FUNCTION_BLOCK FB_System_DLK_951
VAR_INPUT
	Freigabe_auto				: BOOL;
	Freigabe_Deakt_auto			: BOOL;
	Betrieb_Anford_auto			: BOOL;
END_VAR
VAR_OUTPUT
	{attribute 'OPC.UA.DA' := '1'}Steuerung				: ST_System_DLK_Steuerung;		
	{attribute 'OPC.UA.DA' := '1'}Stellwert				: ST_System_DLK_Stellwert;		
	{attribute 'OPC.UA.DA' := '1'}Zustand					: ST_System_DLK_Zustand;	
	{attribute 'OPC.UA.DA' := '1'}Parameter				: ST_System_DLK_Parameter;		
END_VAR
VAR
	Pumpe_251				: FB_PU;
	Stellventil_251			: FB_SVs;
	Regelventil_251			: FB_RV;	(* 14.07.2020*)
	Druckluftkompressor_951	: FB_DLK;

	Zustandscheck			: FB_System_DLK_Zustandscheck;
	Logik					: FB_System_DLK_Logik;
	Ablaufsteuerung			: FB_System_DLK_Ablaufsteuerung;
	Stellwertscheck			: FB_System_DLK_Stellwertscheck;

END_VAR
VAR // added by the converter: edge detectors and wires of the graphical bodies
    _w1 : ANY;
END_VAR

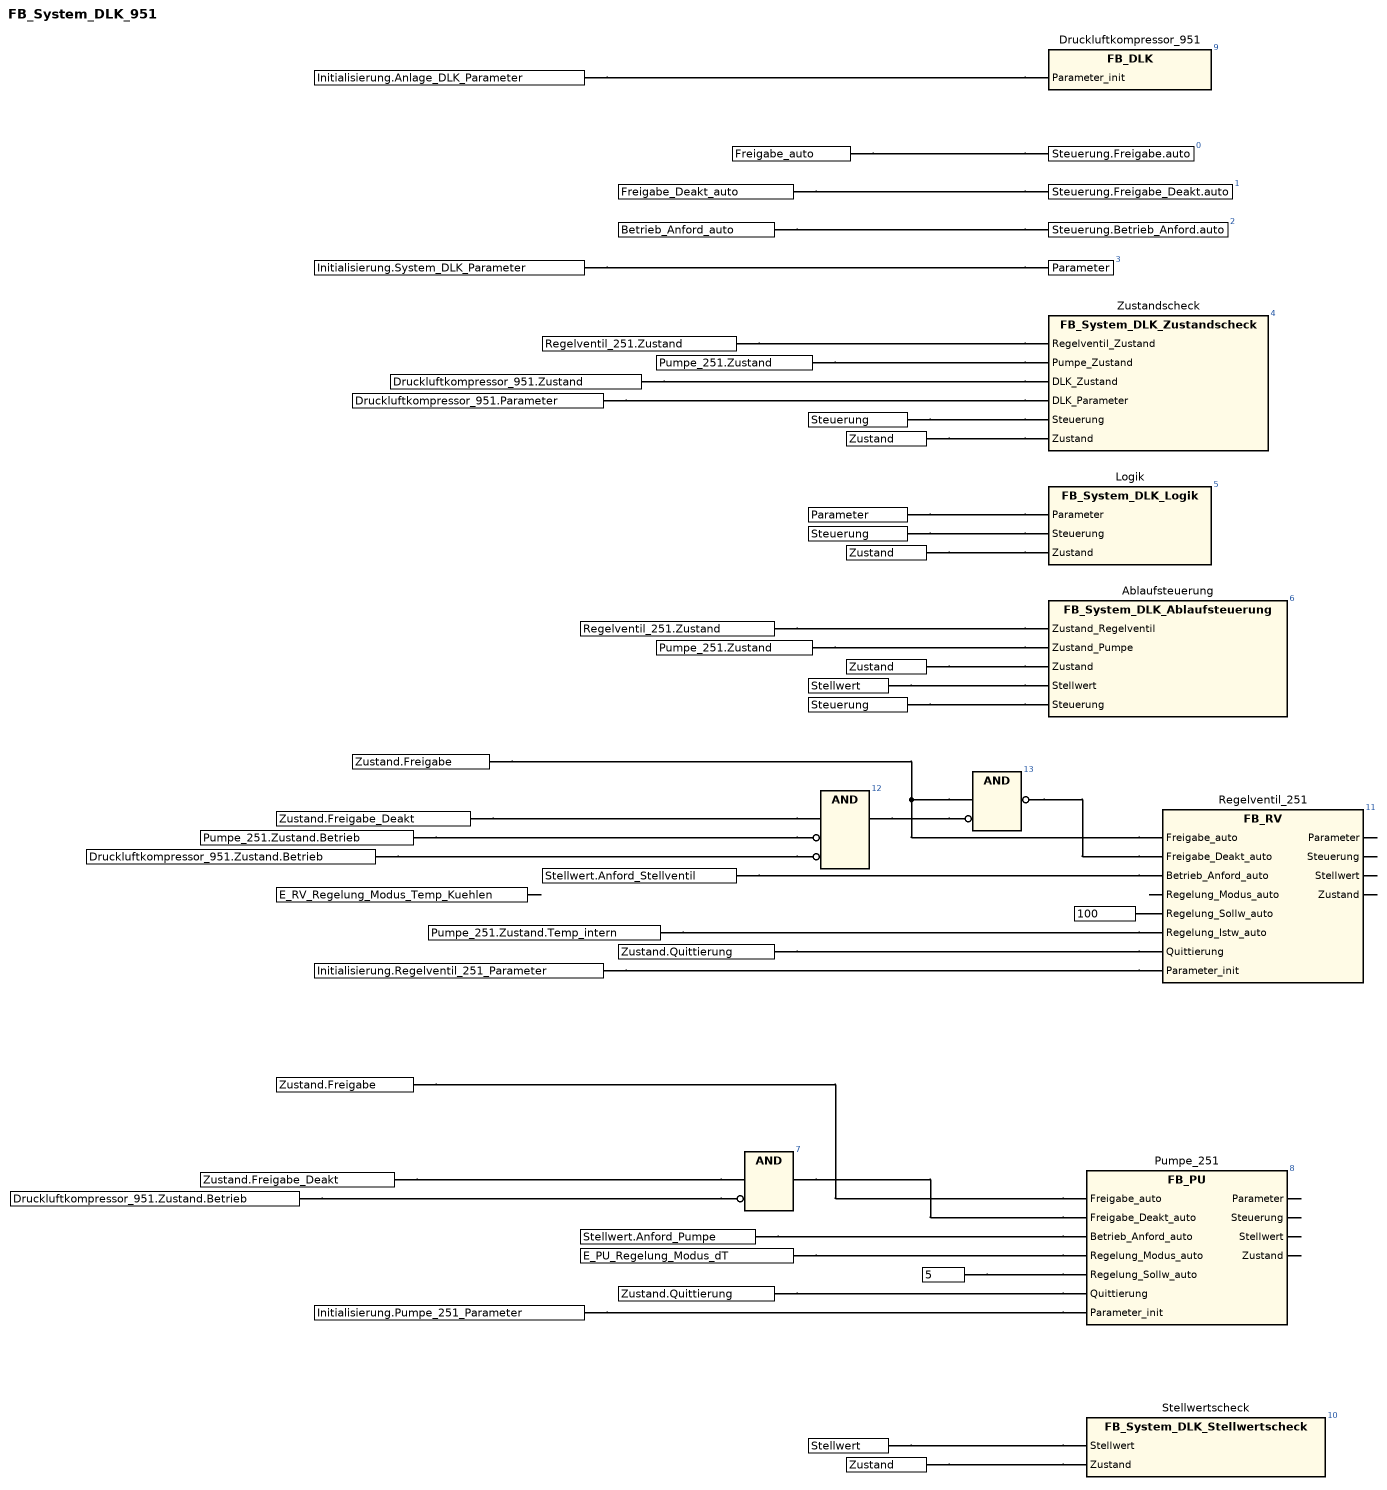
Steuerung.Freigabe.auto := Freigabe_auto;
Steuerung.Freigabe_Deakt.auto := Freigabe_Deakt_auto;
Steuerung.Betrieb_Anford.auto := Betrieb_Anford_auto;
Parameter := Initialisierung.System_DLK_Parameter;
Zustandscheck(
    Regelventil_Zustand := Regelventil_251.Zustand,
    Pumpe_Zustand := Pumpe_251.Zustand,
    DLK_Zustand := Druckluftkompressor_951.Zustand,
    DLK_Parameter := Druckluftkompressor_951.Parameter,
    Steuerung := Steuerung,
    Zustand := Zustand); // FB_System_DLK_Zustandscheck
Logik(Parameter := Parameter, Steuerung := Steuerung, Zustand := Zustand); // FB_System_DLK_Logik
Ablaufsteuerung(
    Zustand_Regelventil := Regelventil_251.Zustand,
    Zustand_Pumpe := Pumpe_251.Zustand,
    Zustand := Zustand,
    Stellwert := Stellwert,
    Steuerung := Steuerung); // FB_System_DLK_Ablaufsteuerung
Pumpe_251(
    Freigabe_auto := Zustand.Freigabe,
    Freigabe_Deakt_auto := Zustand.Freigabe_Deakt AND NOT Druckluftkompressor_951.Zustand.Betrieb,
    Betrieb_Anford_auto := Stellwert.Anford_Pumpe,
    Regelung_Modus_auto := E_PU_Regelung_Modus_dT,
    Regelung_Sollw_auto := 5,
    Quittierung := Zustand.Quittierung,
    Parameter_init := Initialisierung.Pumpe_251_Parameter); // FB_PU
Druckluftkompressor_951(Parameter_init := Initialisierung.Anlage_DLK_Parameter); // FB_DLK
Stellwertscheck(Stellwert := Stellwert, Zustand := Zustand); // FB_System_DLK_Stellwertscheck
Regelventil_251(
    Freigabe_auto := Zustand.Freigabe,
    Freigabe_Deakt_auto := NOT _w1,
    Betrieb_Anford_auto := Stellwert.Anford_Stellventil,
    Regelung_Sollw_auto := 100,
    Regelung_Istw_auto := Pumpe_251.Zustand.Temp_intern,
    Quittierung := Zustand.Quittierung,
    Parameter_init := Initialisierung.Regelventil_251_Parameter); // FB_RV
_w1 := Zustand.Freigabe AND NOT (Zustand.Freigabe_Deakt AND NOT Pumpe_251.Zustand.Betrieb AND NOT Druckluftkompressor_951.Zustand.Betrieb);
// E_RV_Regelung_Modus_Temp_Kuehlen: input not connected

END_FUNCTION_BLOCK

(* stored: Version 1.1.0.1, ProductVersion 3.1.4024.9
   POU FB_System_DLK_951: Id {c935c365-716b-4cef-ac5f-1d94b8db87bf}, SpecialFunc None *)
